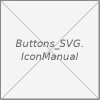
VISUALIZATION ButtonManual  // 100x100
VAR_IN_OUT
	bState : BOOL;
END_VAR
    Frame (0,0 100x100)
        shows ButtonTemplate(bActive := bState)
    Image (0,0 100x100), image: Buttons_SVG.IconManual
        OnMouseDown: execute { GVL_HMI.fbHMIControl.eScreenRequest := E_BaseVisu.Manual; }
END_VISUALIZATION

(* stored: Version 1.1.0.1, ProductVersion 3.1.4024.11
   Visu ButtonManual: Id {ef50f116-a4f8-43e9-b9be-0a50ee093570} *)
